# EPICS substitutions: ek9000App/Db/EL3054.substitutions
file EL3054.template
{       pattern
        {
                TERMINAL,

        }
        {
        }
}
